// ----------------------------------------------------------
// PID01 spare
// ----------------------------------------------------------
// starting value -----------------------
//A     "U130ActD".Act.OutI // !!! insert correct Act !!!
      A     #GenRel;
      CLR   ;
      =     DB5306.DBX  203.2;
      =     DB5306.DBX  203.5;

// enable alarm -------------------------
      A     DB5306.DBX  203.5;
      A     DB5306.DBX  201.4;
      AN    DB5306.DBX  203.1;
      AN    DB5306.DBX  203.3;
      AN    DB5306.DBX  203.4;
      =     DB5306.DBX  203.0;

// setpoint to controller ---------------
      L     DB4301.DBD 1118; // !!! insert correct SFM !!!
      T     DB5306.DBD  234;

// static value to controller ----------
      L     DB4301.DBD 1118; // !!! insert correct SFM !!!
      T     DB5306.DBD  238;

// process value to controller ----------
      L     DB5303.DBD   26; // !!! insert correct AnI !!!
      T     DB5306.DBD  254;

// low/high value to controller ---------
      L     DB5303.DBD   30; // !!! insert correct AnI !!!
      T     DB5306.DBD  218;

      L     DB5303.DBD   34; // !!! insert correct AnI !!!
      T     DB5306.DBD  222;

NETWORK
TITLE =Sequence organisation

      CLR   ;
      =     M    122.2;

// SFM supply ----------------------------------------------------------------

// analog value to SFM spare -----------------------
      L     DB5303.DBD  146;
      T     DB4301.DBD 1122; // !!! insert correct SFM !!!

// analog value to SFM spare -----------------------
      L     DB5303.DBD  266;
      T     DB4301.DBD 1122; // !!! insert correct SFM !!!

// analog value to SFM spare -----------------------
      L     DB5303.DBD  386;
      T     DB4301.DBD 1122; // !!! insert correct SFM !!!

// sequencer ----------------------------------------------------------------
      A     DB4303.DBX   43.1;
      S     DB4303.DBX   97.3;

      CALL FC    40 (
           UnitNo                   := #UnitNo);

NETWORK
TITLE =Auto / Manual

      SET   ;
      AN    M    122.2;
      JC    MODE;
      AN    M    120.1;


// assign PID mode
      S     DB5306.DBX  201.4;
      S     DB5306.DBX  201.5;


MODE: SET   ;

END_FUNCTION_BLOCK

FUNCTION_BLOCK FB 4310
TITLE =U131: Planung Transfer J6F
FAMILY : BOTEC_F1
NAME : U131A
VERSION : 2.1


VAR_TEMP
  EStopOK : BOOL ;	//auxiliary flag
  CIP : BOOL ;	//CIP Program Selected
  xTmp : BOOL ;	//Temporary Bool(free for general use)
  DummyBool : BOOL ;	//Temporary Bool(free for general use)
  UnitNo : INT ;	//unit number
  UnitFB : INT ;	//unit expansion FB number
  rTmp : REAL ;	//Temporary REAL (free for general use)
  iTmp : INT ;	//Temporary INT (free for general use)
  DummyInt : INT ;	//Temporary INT (free for general use)
  dTmp : DINT ;	//Temporary DINT (free for general use)
END_VAR
BEGIN
NETWORK
TITLE =general

      CLR   ;
      =     #xTmp;
      =     #EStopOK;

      L     DB4310.DBW    0;
      T     #UnitNo;
      L     DB4310.DBW    2;
      T     #UnitFB;

NETWORK
TITLE =analog inputs

      NOP   0;
// C_AnI01 AnI 001 spare
      CALL FC    24 (
           UnitNo                   := #UnitNo,
           AnIRec                   := DB5313.C_AnI01,
           ValPer                   := #DummyInt);

// C_AnI002 AnI 002 spare
      CALL FC    24 (
           UnitNo                   := #UnitNo,
           AnIRec                   := DB5313.C_AnI002,
           ValPer                   := #DummyInt);

// AnI03 AnI 003 spare
      CALL FC    24 (
           UnitNo                   := #UnitNo,
           AnIRec                   := DB5313.AnI03,
           ValPer                   := #DummyInt);

NETWORK
TITLE =Universal value

      NOP   0;
// unv001 UnV 001 Process Status
      CALL FC    27 (
           UnitNo                   := #UnitNo,
           UnVRec                   := DB5315.unv001,
           ValExt                   := DB5315.DBD  234);

// unv002 UnV 002 Universal Value 02
      CALL FC    27 (
           UnitNo                   := #UnitNo,
           UnVRec                   := DB5315.unv002,
           ValExt                   := DB5315.DBD  362);

// unv003 UnV 003 Druck Sollwert
      CALL FC    27 (
           UnitNo                   := #UnitNo,
           UnVRec                   := DB5315.unv003,
           ValExt                   := DB5315.DBD  490);

// unv004 UnV 004 Universal Value 04
      CALL FC    27 (
           UnitNo                   := #UnitNo,
           UnVRec                   := DB5315.unv004,
           ValExt                   := DB5315.DBD  618);

NETWORK
TITLE =special inputs

      NOP   0;
// SpI01 SpI 001 spare
      CALL FC    14 (
           UnitNo                   := #UnitNo,
           SpIRec                   := DB5311.SpI01,
           SpIBit                   := #DummyBool);

// SpI02 SpI 002 spare
      CALL FC    14 (
           UnitNo                   := #UnitNo,
           SpIRec                   := DB5311.SpI02,
           SpIBit                   := #DummyBool);

// SpI03 SpI 003 spare
      CALL FC    14 (
           UnitNo                   := #UnitNo,
           SpIRec                   := DB5311.SpI03,
           SpIBit                   := #DummyBool);

// SpI04 SpI 004 spare
      CALL FC    14 (
           UnitNo                   := #UnitNo,
           SpIRec                   := DB5311.SpI04,
           SpIBit                   := #DummyBool);

NETWORK
TITLE =messages

      NOP   0;
// msg001 Msg 001 Message 01
      CALL FC    16 (
           UnitNo                   := #UnitNo,
           MsgRec                   := DB5317.msg001,
           MsgBit                   := DB5317.DBX   82.7);

// msg002 Msg 002 Message 02
      CALL FC    16 (
           UnitNo                   := #UnitNo,
           MsgRec                   := DB5317.msg002,
           MsgBit                   := DB5317.DBX  142.7);

// msg003 Msg 003 Message 03
      CALL FC    16 (
           UnitNo                   := #UnitNo,
           MsgRec                   := DB5317.msg003,
           MsgBit                   := DB5317.DBX  202.7);

NETWORK
TITLE =controllers

      NOP   0;
// PID01 PID 001 spare
      CALL FC    55 (
           UnitNo                   := #UnitNo,
           PIDRec                   := DB5316.PID01,
           SpExt                    := DB5316.DBD  234,
           PVal                     := DB5316.DBD  254,
           OPer                     := #DummyInt);

NETWORK
TITLE =unit supply

      UC    FB [#UnitFB];
END_FUNCTION_BLOCK

FUNCTION_BLOCK FB 4311
TITLE =U131: Planung Transfer J6F
FAMILY : BOTEC_F1
NAME : U131E
VERSION : 1.2


VAR_TEMP
  CIP : BOOL ;	//CIP active
  UNIM : BOOL ;	//Unit Not In Maintenance
  GenRel : BOOL ;	//general OK (emergency and maintenance OK)
  EStopOK : BOOL ;	//emergency OK
  UnitNo : INT ;	//unit number
  xTmp : BOOL ;	//Temporary Bool
  iTmp : INT ;	//Temporary INT
  rTmp : REAL ;	//Temporary REAL
  dTmp : DINT ;	//Temporary DINT (free for general use)
  RetValInt : INT ;	//return value
END_VAR
BEGIN
NETWORK
TITLE =General

      SET   ;
// Simulation ---------------------------------------------------------------
      A     DB4311.DBX 1357.7;
      CC    FB  4319; // "U131Sim"
      A     DB4311.DBX   17.3;
      =     DB4311.DBX 1357.7; //Help bit for simulation

// get unit number ----------------------------------------------------------
      L     DB4310.DBW    0;
      T     #UnitNo;

// CIP ----------------------------------------------------------------------
      L     DB4311.DBD   54;
      L     0;
      <D    ;
      =     #CIP;

// emergency OK -------------------------------------------------------------
      A     DB4315.DBX   27.0; //Emergency Stop OK
      =     #EStopOK;

// Write Unit in Maintenance ------------------------------------------------

      AN    DB4311.DBX   69.7;
      =     #UNIM;

// emergency and maintenance OK ---------------------------------------------
      A     #EStopOK;
      A     #UNIM;
      =     #GenRel;

// communication ------------------------------------------------------------
      UC    FB  4315; // U131Com

NETWORK
TITLE =Analog Inputs

      NOP   0;

// ----------------------------------------------------------
// C_AnI01 spare
// ----------------------------------------------------------
      L     DB4311.DBD 1118; // !!! insert correct SFM !!!
      T     DB5313.DBD  238;

      SET   ;
      =     DB5313.DBX  141.5;

// ----------------------------------------------------------
// C_AnI002 spare
// ----------------------------------------------------------
      L     DB4311.DBD 1118; // !!! insert correct SFM !!!
      T     DB5313.DBD  358;

      SET   ;
      =     DB5313.DBX  261.5;

// ----------------------------------------------------------
// AnI03 spare
// ----------------------------------------------------------
      L     DB4311.DBD 1118; // !!! insert correct SFM !!!
      T     DB5313.DBD  478;

      SET   ;
      =     DB5313.DBX  381.5;

NETWORK
TITLE =Universal Value

      NOP   0;

// ----------------------------------------------------------
// unv001 Process Status
// ----------------------------------------------------------
// process value to UnV
//      L     0.000000e+000
//      T     "U131UnVD".unv001.ValExt

// ----------------------------------------------------------
// unv002 Universal Value 02
// ----------------------------------------------------------
// process value to UnV
//      L     0.000000e+000
//      T     "U131UnVD".unv002.ValExt

// ----------------------------------------------------------
// unv003 Druck Sollwert
// ----------------------------------------------------------
// process value to UnV
//      L     0.000000e+000
//      T     "U131UnVD".unv003.ValExt

// ----------------------------------------------------------
// unv004 Universal Value 04
// ----------------------------------------------------------
// process value to UnV
//      L     0.000000e+000
//      T     "U131UnVD".unv004.ValExt

NETWORK
TITLE =Special Input

      NOP   0;

// ----------------------------------------------------------
// SpI01 spare
// ----------------------------------------------------------
      SET   ;
      =     DB5311.DBX   81.4;
      =     DB5311.DBX   81.5;

// ----------------------------------------------------------
// SpI02 spare
// ----------------------------------------------------------
      SET   ;
      =     DB5311.DBX  141.4;
      =     DB5311.DBX  141.5;

// ----------------------------------------------------------
// SpI03 spare
// ----------------------------------------------------------
      SET   ;
      =     DB5311.DBX  201.4;
      =     DB5311.DBX  201.5;

// ----------------------------------------------------------
// SpI04 spare
// ----------------------------------------------------------
      SET   ;
      =     DB5311.DBX  261.4;
      =     DB5311.DBX  261.5;

NETWORK
TITLE =Messages

      NOP   0;

// ----------------------------------------------------------
// msg001 Message 01
// ----------------------------------------------------------
      SET   ;
      R     DB5317.DBX   80.7;
      =     DB5317.DBX   81.4;

      CLR   ;
      =     DB5317.DBX   82.7;

// ----------------------------------------------------------
// msg002 Message 02
// ----------------------------------------------------------
      SET   ;
      R     DB5317.DBX  140.7;
      =     DB5317.DBX  141.4;

      CLR   ;
      =     DB5317.DBX  142.7;

// ----------------------------------------------------------
// msg003 Message 03
// ----------------------------------------------------------
      SET   ;
      R     DB5317.DBX  200.7;
      =     DB5317.DBX  201.4;

      CLR   ;
      =     DB5317.DBX  202.7;

NETWORK
TITLE =PID controller

      NOP   0;

// ----------------------------------------------------------
// PID01 spare
// ----------------------------------------------------------
// starting value -----------------------
//A     "U131ActD".Act.OutI // !!! insert correct Act !!!
      A     #GenRel;
      CLR   ;
      =     DB5316.DBX  203.2;
      =     DB5316.DBX  203.5;

// enable alarm -------------------------
      A     DB5316.DBX  203.5;
      A     DB5316.DBX  201.4;
      AN    DB5316.DBX  203.1;
      AN    DB5316.DBX  203.3;
      AN    DB5316.DBX  203.4;
      =     DB5316.DBX  203.0;

// setpoint to controller ---------------
      L     DB4311.DBD 1118; // !!! insert correct SFM !!!
      T     DB5316.DBD  234;

// static value to controller ----------
      L     DB4311.DBD 1118; // !!! insert correct SFM !!!
      T     DB5316.DBD  238;

// process value to controller ----------
      L     DB5313.DBD   26; // !!! insert correct AnI !!!
      T     DB5316.DBD  254;

// low/high value to controller ---------
      L     DB5313.DBD   30; // !!! insert correct AnI !!!
      T     DB5316.DBD  218;

      L     DB5313.DBD   34; // !!! insert correct AnI !!!
      T     DB5316.DBD  222;

NETWORK
TITLE =Sequence organisation

      CLR   ;
      =     M    122.2;

// SFM supply ----------------------------------------------------------------

// analog value to SFM spare -----------------------
      L     DB5313.DBD  146;
      T     DB4311.DBD 1122; // !!! insert correct SFM !!!

// analog value to SFM spare -----------------------
      L     DB5313.DBD  266;
      T     DB4311.DBD 1122; // !!! insert correct SFM !!!

// analog value to SFM spare -----------------------
      L     DB5313.DBD  386;
      T     DB4311.DBD 1122; // !!! insert correct SFM !!!

// sequencer ----------------------------------------------------------------
      A     DB4313.DBX   43.1;
      S     DB4313.DBX   97.3;

      CALL FC    40 (
           UnitNo                   := #UnitNo);

NETWORK
TITLE =Auto / Manual

      SET   ;
      AN    M    122.2;
      JC    MODE;
      AN    M    120.1;


// assign PID mode
      S     DB5316.DBX  201.4;
      S     DB5316.DBX  201.5;


MODE: SET   ;

END_FUNCTION_BLOCK

FUNCTION_BLOCK FB 4320
TITLE =U132: Planung Transfer L6F
FAMILY : BOTEC_F1
NAME : U132A
VERSION : 2.1


VAR_TEMP
  EStopOK : BOOL ;	//auxiliary flag
  CIP : BOOL ;	//CIP Program Selected
  xTmp : BOOL ;	//Temporary Bool(free for general use)
  DummyBool : BOOL ;	//Temporary Bool(free for general use)
  UnitNo : INT ;	//unit number
  UnitFB : INT ;	//unit expansion FB number
  rTmp : REAL ;	//Temporary REAL (free for general use)
  iTmp : INT ;	//Temporary INT (free for general use)
  DummyInt : INT ;	//Temporary INT (free for general use)
  dTmp : DINT ;	//Temporary DINT (free for general use)
END_VAR
BEGIN
NETWORK
TITLE =general

      CLR   ;
      =     #xTmp;
      =     #EStopOK;

      L     DB4320.DBW    0;
      T     #UnitNo;
      L     DB4320.DBW    2;
      T     #UnitFB;

NETWORK
TITLE =analog inputs

      NOP   0;
// C_AnI01 AnI 001 spare
      CALL FC    24 (
           UnitNo                   := #UnitNo,
           AnIRec                   := DB5323.C_AnI01,
           ValPer                   := #DummyInt);

// C_AnI002 AnI 002 spare
      CALL FC    24 (
           UnitNo                   := #UnitNo,
           AnIRec                   := DB5323.C_AnI002,
           ValPer                   := #DummyInt);

// AnI03 AnI 003 spare
      CALL FC    24 (
           UnitNo                   := #UnitNo,
           AnIRec                   := DB5323.AnI03,
           ValPer                   := #DummyInt);

NETWORK
TITLE =Universal value

      NOP   0;
// unv001 UnV 001 Process Status
      CALL FC    27 (
           UnitNo                   := #UnitNo,
           UnVRec                   := DB5325.unv001,
           ValExt                   := DB5325.DBD  234);

// unv002 UnV 002 Universal Value 02
      CALL FC    27 (
           UnitNo                   := #UnitNo,
           UnVRec                   := DB5325.unv002,
           ValExt                   := DB5325.DBD  362);

// unv003 UnV 003 Druck Sollwert
      CALL FC    27 (
           UnitNo                   := #UnitNo,
           UnVRec                   := DB5325.unv003,
           ValExt                   := DB5325.DBD  490);

// unv004 UnV 004 Universal Value 04
      CALL FC    27 (
           UnitNo                   := #UnitNo,
           UnVRec                   := DB5325.unv004,
           ValExt                   := DB5325.DBD  618);

NETWORK
TITLE =special inputs

      NOP   0;
// SpI01 SpI 001 spare
      CALL FC    14 (
           UnitNo                   := #UnitNo,
           SpIRec                   := DB5321.SpI01,
           SpIBit                   := #DummyBool);

// SpI02 SpI 002 spare
      CALL FC    14 (
           UnitNo                   := #UnitNo,
           SpIRec                   := DB5321.SpI02,
           SpIBit                   := #DummyBool);

// SpI03 SpI 003 spare
      CALL FC    14 (
           UnitNo                   := #UnitNo,
           SpIRec                   := DB5321.SpI03,
           SpIBit                   := #DummyBool);

// SpI04 SpI 004 spare
      CALL FC    14 (
           UnitNo                   := #UnitNo,
           SpIRec                   := DB5321.SpI04,
           SpIBit                   := #DummyBool);

NETWORK
TITLE =messages

      NOP   0;
// msg001 Msg 001 Message 01
      CALL FC    16 (
           UnitNo                   := #UnitNo,
           MsgRec                   := DB5327.msg001,
           MsgBit                   := DB5327.DBX   82.7);

// msg002 Msg 002 Message 02
      CALL FC    16 (
           UnitNo                   := #UnitNo,
           MsgRec                   := DB5327.msg002,
           MsgBit                   := DB5327.DBX  142.7);

// msg003 Msg 003 Message 03
      CALL FC    16 (
           UnitNo                   := #UnitNo,
           MsgRec                   := DB5327.msg003,
           MsgBit                   := DB5327.DBX  202.7);

NETWORK
TITLE =controllers

      NOP   0;
// PID01 PID 001 spare
      CALL FC    55 (
           UnitNo                   := #UnitNo,
           PIDRec                   := DB5326.PID01,
           SpExt                    := DB5326.DBD  234,
           PVal                     := DB5326.DBD  254,
           OPer                     := #DummyInt);

NETWORK
TITLE =unit supply

      UC    FB [#UnitFB];
END_FUNCTION_BLOCK

FUNCTION_BLOCK FB 4321
TITLE =U132: Planung Transfer L6F
FAMILY : BOTEC_F1
NAME : U132E
VERSION : 1.2


VAR_TEMP
  CIP : BOOL ;	//CIP active
  UNIM : BOOL ;	//Unit Not In Maintenance
  GenRel : BOOL ;	//general OK (emergency and maintenance OK)
  EStopOK : BOOL ;	//emergency OK
  UnitNo : INT ;	//unit number
  xTmp : BOOL ;	//Temporary Bool
  iTmp : INT ;	//Temporary INT
  rTmp : REAL ;	//Temporary REAL
  dTmp : DINT ;	//Temporary DINT (free for general use)
  RetValInt : INT ;	//return value
END_VAR
BEGIN
NETWORK
TITLE =General

      SET   ;
// Simulation ---------------------------------------------------------------
      A     DB4321.DBX 1357.7;
      CC    FB  4329; // "U132Sim"
      A     DB4321.DBX   17.3;
      =     DB4321.DBX 1357.7; //Help bit for simulation

// get unit number ----------------------------------------------------------
      L     DB4320.DBW    0;
      T     #UnitNo;

// CIP ----------------------------------------------------------------------
      L     DB4321.DBD   54;
      L     0;
      <D    ;
      =     #CIP;

// emergency OK -------------------------------------------------------------
      A     DB4325.DBX   27.0; //Emergency Stop OK
      =     #EStopOK;

// Write Unit in Maintenance ------------------------------------------------

      AN    DB4321.DBX   69.7;
      =     #UNIM;

// emergency and maintenance OK ---------------------------------------------
      A     #EStopOK;
      A     #UNIM;
      =     #GenRel;

// communication ------------------------------------------------------------
      UC    FB  4325; // U132Com

NETWORK
TITLE =Analog Inputs

      NOP   0;

// ----------------------------------------------------------
// C_AnI01 spare
// ----------------------------------------------------------
      L     DB4321.DBD 1118; // !!! insert correct SFM !!!
      T     DB5323.DBD  238;

      SET   ;
      =     DB5323.DBX  141.5;

// ----------------------------------------------------------
// C_AnI002 spare
// ----------------------------------------------------------
      L     DB4321.DBD 1118; // !!! insert correct SFM !!!
      T     DB5323.DBD  358;

      SET   ;
      =     DB5323.DBX  261.5;

// ----------------------------------------------------------
// AnI03 spare
// ----------------------------------------------------------
      L     DB4321.DBD 1118; // !!! insert correct SFM !!!
      T     DB5323.DBD  478;

      SET   ;
      =     DB5323.DBX  381.5;

NETWORK
TITLE =Universal Value

      NOP   0;

// ----------------------------------------------------------
// unv001 Process Status
// ----------------------------------------------------------
// process value to UnV
//      L     0.000000e+000
//      T     "U132UnVD".unv001.ValExt

// ----------------------------------------------------------
// unv002 Universal Value 02
// ----------------------------------------------------------
// process value to UnV
//      L     0.000000e+000
//      T     "U132UnVD".unv002.ValExt

// ----------------------------------------------------------
// unv003 Druck Sollwert
// ----------------------------------------------------------
// process value to UnV
//      L     0.000000e+000
//      T     "U132UnVD".unv003.ValExt

// ----------------------------------------------------------
// unv004 Universal Value 04
// ----------------------------------------------------------
// process value to UnV
//      L     0.000000e+000
//      T     "U132UnVD".unv004.ValExt

NETWORK
TITLE =Special Input

      NOP   0;

// ----------------------------------------------------------
// SpI01 spare
// ----------------------------------------------------------
      SET   ;
      =     DB5321.DBX   81.4;
      =     DB5321.DBX   81.5;

// ----------------------------------------------------------
// SpI02 spare
// ----------------------------------------------------------
      SET   ;
      =     DB5321.DBX  141.4;
      =     DB5321.DBX  141.5;

// ----------------------------------------------------------
// SpI03 spare
// ----------------------------------------------------------
      SET   ;
      =     DB5321.DBX  201.4;
      =     DB5321.DBX  201.5;

// ----------------------------------------------------------
// SpI04 spare
// ----------------------------------------------------------
      SET   ;
      =     DB5321.DBX  261.4;
      =     DB5321.DBX  261.5;

NETWORK
TITLE =Messages

      NOP   0;

// ----------------------------------------------------------
// msg001 Message 01
// ----------------------------------------------------------
      SET   ;
      R     DB5327.DBX   80.7;
      =     DB5327.DBX   81.4;

      CLR   ;
      =     DB5327.DBX   82.7;

// ----------------------------------------------------------
// msg002 Message 02
// ----------------------------------------------------------
      SET   ;
      R     DB5327.DBX  140.7;
      =     DB5327.DBX  141.4;

      CLR   ;
      =     DB5327.DBX  142.7;

// ----------------------------------------------------------
// msg003 Message 03
// ----------------------------------------------------------
      SET   ;
      R     DB5327.DBX  200.7;
      =     DB5327.DBX  201.4;

      CLR   ;
      =     DB5327.DBX  202.7;

NETWORK
TITLE =PID controller

      NOP   0;

// ----------------------------------------------------------
// PID01 spare
// ----------------------------------------------------------
// starting value -----------------------
//A     "U132ActD".Act.OutI // !!! insert correct Act !!!
      A     #GenRel;
      CLR   ;
      =     DB5326.DBX  203.2;
      =     DB5326.DBX  203.5;

// enable alarm -------------------------
      A     DB5326.DBX  203.5;
      A     DB5326.DBX  201.4;
      AN    DB5326.DBX  203.1;
      AN    DB5326.DBX  203.3;
      AN    DB5326.DBX  203.4;
      =     DB5326.DBX  203.0;

// setpoint to controller ---------------
      L     DB4321.DBD 1118; // !!! insert correct SFM !!!
      T     DB5326.DBD  234;

// static value to controller ----------
      L     DB4321.DBD 1118; // !!! insert correct SFM !!!
      T     DB5326.DBD  238;

// process value to controller ----------
      L     DB5323.DBD   26; // !!! insert correct AnI !!!
      T     DB5326.DBD  254;

// low/high value to controller ---------
      L     DB5323.DBD   30; // !!! insert correct AnI !!!
      T     DB5326.DBD  218;

      L     DB5323.DBD   34; // !!! insert correct AnI !!!
      T     DB5326.DBD  222;

NETWORK
TITLE =Sequence organisation

      CLR   ;
      =     M    122.2;

// SFM supply ----------------------------------------------------------------

// analog value to SFM spare -----------------------
      L     DB5323.DBD  146;
      T     DB4321.DBD 1122; // !!! insert correct SFM !!!

// analog value to SFM spare -----------------------
      L     DB5323.DBD  266;
      T     DB4321.DBD 1122; // !!! insert correct SFM !!!

// analog value to SFM spare -----------------------
      L     DB5323.DBD  386;
      T     DB4321.DBD 1122; // !!! insert correct SFM !!!

// sequencer ----------------------------------------------------------------
      A     DB4323.DBX   43.1;
      S     DB4323.DBX   97.3;

      CALL FC    40 (
           UnitNo                   := #UnitNo);

NETWORK
TITLE =Auto / Manual

      SET   ;
      AN    M    122.2;
      JC    MODE;
      AN    M    120.1;


// assign PID mode
      S     DB5326.DBX  201.4;
      S     DB5326.DBX  201.5;


MODE: SET   ;

END_FUNCTION_BLOCK

FUNCTION_BLOCK FB 4330
TITLE =U133: Planung Transfer B6
FAMILY : BOTEC_F1
NAME : U133A
VERSION : 2.1


VAR_TEMP
  EStopOK : BOOL ;	//auxiliary flag
  CIP : BOOL ;	//CIP Program Selected
  xTmp : BOOL ;	//Temporary Bool(free for general use)
  DummyBool : BOOL ;	//Temporary Bool(free for general use)
  UnitNo : INT ;	//unit number
  UnitFB : INT ;	//unit expansion FB number
  rTmp : REAL ;	//Temporary REAL (free for general use)
  iTmp : INT ;	//Temporary INT (free for general use)
  DummyInt : INT ;	//Temporary INT (free for general use)
  dTmp : DINT ;	//Temporary DINT (free for general use)
END_VAR
BEGIN
NETWORK
TITLE =general

      CLR   ;
      =     #xTmp;
      =     #EStopOK;

      L     DB4330.DBW    0;
      T     #UnitNo;
      L     DB4330.DBW    2;
      T     #UnitFB;

NETWORK
TITLE =analog inputs

      NOP   0;
// C_AnI01 AnI 001 spare
      CALL FC    24 (
           UnitNo                   := #UnitNo,
           AnIRec                   := DB5333.C_AnI01,
           ValPer                   := #DummyInt);

// C_AnI002 AnI 002 spare
      CALL FC    24 (
           UnitNo                   := #UnitNo,
           AnIRec                   := DB5333.C_AnI002,
           ValPer                   := #DummyInt);

// AnI03 AnI 003 spare
      CALL FC    24 (
           UnitNo                   := #UnitNo,
           AnIRec                   := DB5333.AnI03,
           ValPer                   := #DummyInt);

NETWORK
TITLE =Universal value

      NOP   0;
// unv001 UnV 001 Process Status
      CALL FC    27 (
           UnitNo                   := #UnitNo,
           UnVRec                   := DB5335.unv001,
           ValExt                   := DB5335.DBD  234);

// unv002 UnV 002 Universal Value 02
      CALL FC    27 (
           UnitNo                   := #UnitNo,
           UnVRec                   := DB5335.unv002,
           ValExt                   := DB5335.DBD  362);

// unv003 UnV 003 Druck Sollwert
      CALL FC    27 (
           UnitNo                   := #UnitNo,
           UnVRec                   := DB5335.unv003,
           ValExt                   := DB5335.DBD  490);

// unv004 UnV 004 Universal Value 04
      CALL FC    27 (
           UnitNo                   := #UnitNo,
           UnVRec                   := DB5335.unv004,
           ValExt                   := DB5335.DBD  618);

NETWORK
TITLE =special inputs

      NOP   0;
// SpI01 SpI 001 spare
      CALL FC    14 (
           UnitNo                   := #UnitNo,
           SpIRec                   := DB5331.SpI01,
           SpIBit                   := #DummyBool);

// SpI02 SpI 002 spare
      CALL FC    14 (
           UnitNo                   := #UnitNo,
           SpIRec                   := DB5331.SpI02,
           SpIBit                   := #DummyBool);

// SpI03 SpI 003 spare
      CALL FC    14 (
           UnitNo                   := #UnitNo,
           SpIRec                   := DB5331.SpI03,
           SpIBit                   := #DummyBool);

// SpI04 SpI 004 spare
      CALL FC    14 (
           UnitNo                   := #UnitNo,
           SpIRec                   := DB5331.SpI04,
           SpIBit                   := #DummyBool);

NETWORK
TITLE =messages

      NOP   0;
// msg001 Msg 001 Message 01
      CALL FC    16 (
           UnitNo                   := #UnitNo,
           MsgRec                   := DB5337.msg001,
           MsgBit                   := DB5337.DBX   82.7);

// msg002 Msg 002 Message 02
      CALL FC    16 (
           UnitNo                   := #UnitNo,
           MsgRec                   := DB5337.msg002,
           MsgBit                   := DB5337.DBX  142.7);

// msg003 Msg 003 Message 03
      CALL FC    16 (
           UnitNo                   := #UnitNo,
           MsgRec                   := DB5337.msg003,
           MsgBit                   := DB5337.DBX  202.7);

NETWORK
TITLE =controllers

      NOP   0;
// PID01 PID 001 spare
      CALL FC    55 (
           UnitNo                   := #UnitNo,
           PIDRec                   := DB5336.PID01,
           SpExt                    := DB5336.DBD  234,
           PVal                     := DB5336.DBD  254,
           OPer                     := #DummyInt);

NETWORK
TITLE =unit supply

      UC    FB [#UnitFB];
END_FUNCTION_BLOCK

FUNCTION_BLOCK FB 4331
TITLE =U133: Planung Transfer B6
FAMILY : BOTEC_F1
NAME : U133E
VERSION : 1.2


VAR_TEMP
  CIP : BOOL ;	//CIP active
  UNIM : BOOL ;	//Unit Not In Maintenance
  GenRel : BOOL ;	//general OK (emergency and maintenance OK)
  EStopOK : BOOL ;	//emergency OK
  UnitNo : INT ;	//unit number
  xTmp : BOOL ;	//Temporary Bool
  iTmp : INT ;	//Temporary INT
  rTmp : REAL ;	//Temporary REAL
  dTmp : DINT ;	//Temporary DINT (free for general use)
  RetValInt : INT ;	//return value
END_VAR
BEGIN
NETWORK
TITLE =General

      SET   ;
// Simulation ---------------------------------------------------------------
      A     DB4331.DBX 1357.7;
      CC    FB  4339; // "U133Sim"
      A     DB4331.DBX   17.3;
      =     DB4331.DBX 1357.7; //Help bit for simulation

// get unit number ----------------------------------------------------------
      L     DB4330.DBW    0;
      T     #UnitNo;

// CIP ----------------------------------------------------------------------
      L     DB4331.DBD   54;
      L     0;
      <D    ;
      =     #CIP;

// emergency OK -------------------------------------------------------------
      A     DB4335.DBX   27.0; //Emergency Stop OK
      =     #EStopOK;

// Write Unit in Maintenance ------------------------------------------------

      AN    DB4331.DBX   69.7;
      =     #UNIM;

// emergency and maintenance OK ---------------------------------------------
      A     #EStopOK;
      A     #UNIM;
      =     #GenRel;

// communication ------------------------------------------------------------
      UC    FB  4335; // U133Com

NETWORK
TITLE =Analog Inputs

      NOP   0;

// ----------------------------------------------------------
// C_AnI01 spare
// ----------------------------------------------------------
      L     DB4331.DBD 1118; // !!! insert correct SFM !!!
      T     DB5333.DBD  238;

      SET   ;
      =     DB5333.DBX  141.5;

// ----------------------------------------------------------
// C_AnI002 spare
// ----------------------------------------------------------
      L     DB4331.DBD 1118; // !!! insert correct SFM !!!
      T     DB5333.DBD  358;

      SET   ;
      =     DB5333.DBX  261.5;

// ----------------------------------------------------------
// AnI03 spare
// ----------------------------------------------------------
      L     DB4331.DBD 1118; // !!! insert correct SFM !!!
      T     DB5333.DBD  478;

      SET   ;
      =     DB5333.DBX  381.5;

NETWORK
TITLE =Universal Value

      NOP   0;

// ----------------------------------------------------------
// unv001 Process Status
// ----------------------------------------------------------
// process value to UnV
//      L     0.000000e+000
//      T     "U133UnVD".unv001.ValExt

// ----------------------------------------------------------
// unv002 Universal Value 02
// ----------------------------------------------------------
// process value to UnV
//      L     0.000000e+000
//      T     "U133UnVD".unv002.ValExt

// ----------------------------------------------------------
// unv003 Druck Sollwert
// ----------------------------------------------------------
// process value to UnV
//      L     0.000000e+000
//      T     "U133UnVD".unv003.ValExt

// ----------------------------------------------------------
// unv004 Universal Value 04
// ----------------------------------------------------------
// process value to UnV
//      L     0.000000e+000
//      T     "U133UnVD".unv004.ValExt

NETWORK
TITLE =Special Input

      NOP   0;

// ----------------------------------------------------------
// SpI01 spare
// ----------------------------------------------------------
      SET   ;
      =     DB5331.DBX   81.4;
      =     DB5331.DBX   81.5;

// ----------------------------------------------------------
// SpI02 spare
// ----------------------------------------------------------
      SET   ;
      =     DB5331.DBX  141.4;
      =     DB5331.DBX  141.5;

// ----------------------------------------------------------
// SpI03 spare
// ----------------------------------------------------------
      SET   ;
      =     DB5331.DBX  201.4;
      =     DB5331.DBX  201.5;

// ----------------------------------------------------------
// SpI04 spare
// ----------------------------------------------------------
      SET   ;
      =     DB5331.DBX  261.4;
      =     DB5331.DBX  261.5;

NETWORK
TITLE =Messages

      NOP   0;

// ----------------------------------------------------------
// msg001 Message 01
// ----------------------------------------------------------
      SET   ;
      R     DB5337.DBX   80.7;
      =     DB5337.DBX   81.4;

      CLR   ;
      =     DB5337.DBX   82.7;

// ----------------------------------------------------------
// msg002 Message 02
// ----------------------------------------------------------
      SET   ;
      R     DB5337.DBX  140.7;
      =     DB5337.DBX  141.4;

      CLR   ;
      =     DB5337.DBX  142.7;

// ----------------------------------------------------------
// msg003 Message 03
// ----------------------------------------------------------
      SET   ;
      R     DB5337.DBX  200.7;
      =     DB5337.DBX  201.4;

      CLR   ;
      =     DB5337.DBX  202.7;

NETWORK
TITLE =PID controller

      NOP   0;

// ----------------------------------------------------------
// PID01 spare
// ----------------------------------------------------------
// starting value -----------------------
//A     "U133ActD".Act.OutI // !!! insert correct Act !!!
      A     #GenRel;
      CLR   ;
      =     DB5336.DBX  203.2;
      =     DB5336.DBX  203.5;

// enable alarm -------------------------
      A     DB5336.DBX  203.5;
      A     DB5336.DBX  201.4;
      AN    DB5336.DBX  203.1;
      AN    DB5336.DBX  203.3;
      AN    DB5336.DBX  203.4;
      =     DB5336.DBX  203.0;

// setpoint to controller ---------------
      L     DB4331.DBD 1118; // !!! insert correct SFM !!!
      T     DB5336.DBD  234;

// static value to controller ----------
      L     DB4331.DBD 1118; // !!! insert correct SFM !!!
      T     DB5336.DBD  238;

// process value to controller ----------
      L     DB5333.DBD   26; // !!! insert correct AnI !!!
      T     DB5336.DBD  254;

// low/high value to controller ---------
      L     DB5333.DBD   30; // !!! insert correct AnI !!!
      T     DB5336.DBD  218;

      L     DB5333.DBD   34; // !!! insert correct AnI !!!
      T     DB5336.DBD  222;

NETWORK
TITLE =Sequence organisation

      CLR   ;
      =     M    122.2;

// SFM supply ----------------------------------------------------------------

// analog value to SFM spare -----------------------
      L     DB5333.DBD  146;
      T     DB4331.DBD 1122; // !!! insert correct SFM !!!

// analog value to SFM spare -----------------------
      L     DB5333.DBD  266;
      T     DB4331.DBD 1122; // !!! insert correct SFM !!!

// analog value to SFM spare -----------------------
      L     DB5333.DBD  386;
      T     DB4331.DBD 1122; // !!! insert correct SFM !!!

// sequencer ----------------------------------------------------------------
      A     DB4333.DBX   43.1;
      S     DB4333.DBX   97.3;

      CALL FC    40 (
           UnitNo                   := #UnitNo);

NETWORK
TITLE =Auto / Manual

      SET   ;
      AN    M    122.2;
      JC    MODE;
      AN    M    120.1;


// assign PID mode
      S     DB5336.DBX  201.4;
      S     DB5336.DBX  201.5;


MODE: SET   ;

END_FUNCTION_BLOCK

FUNCTION_BLOCK FB 4340
TITLE =U134: Planung Transfer D6
FAMILY : BOTEC_F1
NAME : U134A
VERSION : 2.1


VAR_TEMP
  EStopOK : BOOL ;	//auxiliary flag
  CIP : BOOL ;	//CIP Program Selected
  xTmp : BOOL ;	//Temporary Bool(free for general use)
  DummyBool : BOOL ;	//Temporary Bool(free for general use)
  UnitNo : INT ;	//unit number
  UnitFB : INT ;	//unit expansion FB number
  rTmp : REAL ;	//Temporary REAL (free for general use)
  iTmp : INT ;	//Temporary INT (free for general use)
  DummyInt : INT ;	//Temporary INT (free for general use)
  dTmp : DINT ;	//Temporary DINT (free for general use)
END_VAR
BEGIN
NETWORK
TITLE =general

      CLR   ;
      =     #xTmp;
      =     #EStopOK;

      L     DB4340.DBW    0;
      T     #UnitNo;
      L     DB4340.DBW    2;
      T     #UnitFB;

NETWORK
TITLE =analog inputs

      NOP   0;
// C_AnI01 AnI 001 spare
      CALL FC    24 (
           UnitNo                   := #UnitNo,
           AnIRec                   := DB5343.C_AnI01,
           ValPer                   := #DummyInt);

// C_AnI002 AnI 002 spare
      CALL FC    24 (
           UnitNo                   := #UnitNo,
           AnIRec                   := DB5343.C_AnI002,
           ValPer                   := #DummyInt);

// AnI03 AnI 003 spare
      CALL FC    24 (
           UnitNo                   := #UnitNo,
           AnIRec                   := DB5343.AnI03,
           ValPer                   := #DummyInt);

NETWORK
TITLE =Universal value

      NOP   0;
// unv001 UnV 001 Process Status
      CALL FC    27 (
           UnitNo                   := #UnitNo,
           UnVRec                   := DB5345.unv001,
           ValExt                   := DB5345.DBD  234);

// unv002 UnV 002 Universal Value 02
      CALL FC    27 (
           UnitNo                   := #UnitNo,
           UnVRec                   := DB5345.unv002,
           ValExt                   := DB5345.DBD  362);

// unv003 UnV 003 Druck Sollwert
      CALL FC    27 (
           UnitNo                   := #UnitNo,
           UnVRec                   := DB5345.unv003,
           ValExt                   := DB5345.DBD  490);

// unv004 UnV 004 Universal Value 04
      CALL FC    27 (
           UnitNo                   := #UnitNo,
           UnVRec                   := DB5345.unv004,
           ValExt                   := DB5345.DBD  618);

NETWORK
TITLE =special inputs

      NOP   0;
// SpI01 SpI 001 spare
      CALL FC    14 (
           UnitNo                   := #UnitNo,
           SpIRec                   := DB5341.SpI01,
           SpIBit                   := #DummyBool);

// SpI02 SpI 002 spare
      CALL FC    14 (
           UnitNo                   := #UnitNo,
           SpIRec                   := DB5341.SpI02,
           SpIBit                   := #DummyBool);

// SpI03 SpI 003 spare
      CALL FC    14 (
           UnitNo                   := #UnitNo,
           SpIRec                   := DB5341.SpI03,
           SpIBit                   := #DummyBool);

// SpI04 SpI 004 spare
      CALL FC    14 (
           UnitNo                   := #UnitNo,
           SpIRec                   := DB5341.SpI04,
           SpIBit                   := #DummyBool);

NETWORK
TITLE =messages

      NOP   0;
// msg001 Msg 001 Message 01
      CALL FC    16 (
           UnitNo                   := #UnitNo,
           MsgRec                   := DB5347.msg001,
           MsgBit                   := DB5347.DBX   82.7);

// msg002 Msg 002 Message 02
      CALL FC    16 (
           UnitNo                   := #UnitNo,
           MsgRec                   := DB5347.msg002,
           MsgBit                   := DB5347.DBX  142.7);

// msg003 Msg 003 Message 03
      CALL FC    16 (
           UnitNo                   := #UnitNo,
           MsgRec                   := DB5347.msg003,
           MsgBit                   := DB5347.DBX  202.7);

NETWORK
TITLE =controllers

      NOP   0;
// PID01 PID 001 spare
      CALL FC    55 (
           UnitNo                   := #UnitNo,
           PIDRec                   := DB5346.PID01,
           SpExt                    := DB5346.DBD  234,
           PVal                     := DB5346.DBD  254,
           OPer                     := #DummyInt);

NETWORK
TITLE =unit supply

      UC    FB [#UnitFB];
END_FUNCTION_BLOCK

FUNCTION_BLOCK FB 4341
TITLE =U134: Planung Transfer D6
FAMILY : BOTEC_F1
NAME : U134E
VERSION : 1.2


VAR_TEMP
  CIP : BOOL ;	//CIP active
  UNIM : BOOL ;	//Unit Not In Maintenance
  GenRel : BOOL ;	//general OK (emergency and maintenance OK)
  EStopOK : BOOL ;	//emergency OK
  UnitNo : INT ;	//unit number
  xTmp : BOOL ;	//Temporary Bool
  iTmp : INT ;	//Temporary INT
  rTmp : REAL ;	//Temporary REAL
  dTmp : DINT ;	//Temporary DINT (free for general use)
  RetValInt : INT ;	//return value
END_VAR
BEGIN
NETWORK
TITLE =General

      SET   ;
// Simulation ---------------------------------------------------------------
      A     DB4341.DBX 1357.7;
      CC    FB  4349; // "U134Sim"
      A     DB4341.DBX   17.3;
      =     DB4341.DBX 1357.7; //Help bit for simulation

// get unit number ----------------------------------------------------------
      L     DB4340.DBW    0;
      T     #UnitNo;

// CIP ----------------------------------------------------------------------
      L     DB4341.DBD   54;
      L     0;
      <D    ;
      =     #CIP;

// emergency OK -------------------------------------------------------------
      A     DB4345.DBX   27.0; //Emergency Stop OK
      =     #EStopOK;

// Write Unit in Maintenance ------------------------------------------------

      AN    DB4341.DBX   69.7;
      =     #UNIM;

// emergency and maintenance OK ---------------------------------------------
      A     #EStopOK;
      A     #UNIM;
      =     #GenRel;

// communication ------------------------------------------------------------
      UC    FB  4345; // U134Com

NETWORK
TITLE =Analog Inputs

      NOP   0;

// ----------------------------------------------------------
// C_AnI01 spare
// ----------------------------------------------------------
      L     DB4341.DBD 1118; // !!! insert correct SFM !!!
      T     DB5343.DBD  238;

      SET   ;
      =     DB5343.DBX  141.5;

// ----------------------------------------------------------
// C_AnI002 spare
// ----------------------------------------------------------
      L     DB4341.DBD 1118; // !!! insert correct SFM !!!
      T     DB5343.DBD  358;

      SET   ;
      =     DB5343.DBX  261.5;

// ----------------------------------------------------------
// AnI03 spare
// ----------------------------------------------------------
      L     DB4341.DBD 1118; // !!! insert correct SFM !!!
      T     DB5343.DBD  478;

      SET   ;
      =     DB5343.DBX  381.5;

NETWORK
TITLE =Universal Value

      NOP   0;

// ----------------------------------------------------------
// unv001 Process Status
// ----------------------------------------------------------
// process value to UnV
//      L     0.000000e+000
//      T     "U134UnVD".unv001.ValExt

// ----------------------------------------------------------
// unv002 Universal Value 02
// ----------------------------------------------------------
// process value to UnV
//      L     0.000000e+000
//      T     "U134UnVD".unv002.ValExt

// ----------------------------------------------------------
// unv003 Druck Sollwert
// ----------------------------------------------------------
// process value to UnV
//      L     0.000000e+000
//      T     "U134UnVD".unv003.ValExt

// ----------------------------------------------------------
// unv004 Universal Value 04
// ----------------------------------------------------------
// process value to UnV
//      L     0.000000e+000
//      T     "U134UnVD".unv004.ValExt

NETWORK
TITLE =Special Input

      NOP   0;

// ----------------------------------------------------------
// SpI01 spare
// ----------------------------------------------------------
      SET   ;
      =     DB5341.DBX   81.4;
      =     DB5341.DBX   81.5;

// ----------------------------------------------------------
// SpI02 spare
// ----------------------------------------------------------
      SET   ;
      =     DB5341.DBX  141.4;
      =     DB5341.DBX  141.5;

// ----------------------------------------------------------
// SpI03 spare
// ----------------------------------------------------------
      SET   ;
      =     DB5341.DBX  201.4;
      =     DB5341.DBX  201.5;

// ----------------------------------------------------------
// SpI04 spare
// ----------------------------------------------------------
      SET   ;
      =     DB5341.DBX  261.4;
      =     DB5341.DBX  261.5;

NETWORK
TITLE =Messages

      NOP   0;

// ----------------------------------------------------------
// msg001 Message 01
// ----------------------------------------------------------
      SET   ;
      R     DB5347.DBX   80.7;
      =     DB5347.DBX   81.4;

      CLR   ;
      =     DB5347.DBX   82.7;

// ----------------------------------------------------------
// msg002 Message 02
// ----------------------------------------------------------
      SET   ;
      R     DB5347.DBX  140.7;
      =     DB5347.DBX  141.4;

      CLR   ;
      =     DB5347.DBX  142.7;

// ----------------------------------------------------------
// msg003 Message 03
// ----------------------------------------------------------
      SET   ;
      R     DB5347.DBX  200.7;
      =     DB5347.DBX  201.4;

      CLR   ;
      =     DB5347.DBX  202.7;

NETWORK
TITLE =PID controller

      NOP   0;

// ----------------------------------------------------------
// PID01 spare
// ----------------------------------------------------------
// starting value -----------------------
//A     "U134ActD".Act.OutI // !!! insert correct Act !!!
      A     #GenRel;
      CLR   ;
      =     DB5346.DBX  203.2;
      =     DB5346.DBX  203.5;

// enable alarm -------------------------
      A     DB5346.DBX  203.5;
      A     DB5346.DBX  201.4;
      AN    DB5346.DBX  203.1;
      AN    DB5346.DBX  203.3;
      AN    DB5346.DBX  203.4;
      =     DB5346.DBX  203.0;

// setpoint to controller ---------------
      L     DB4341.DBD 1118; // !!! insert correct SFM !!!
      T     DB5346.DBD  234;

// static value to controller ----------
      L     DB4341.DBD 1118; // !!! insert correct SFM !!!
      T     DB5346.DBD  238;

// process value to controller ----------
      L     DB5343.DBD   26; // !!! insert correct AnI !!!
      T     DB5346.DBD  254;

// low/high value to controller ---------
      L     DB5343.DBD   30; // !!! insert correct AnI !!!
      T     DB5346.DBD  218;

      L     DB5343.DBD   34; // !!! insert correct AnI !!!
      T     DB5346.DBD  222;

NETWORK
TITLE =Sequence organisation

      CLR   ;
      =     M    122.2;

// SFM supply ----------------------------------------------------------------

// analog value to SFM spare -----------------------
      L     DB5343.DBD  146;
      T     DB4341.DBD 1122; // !!! insert correct SFM !!!

// analog value to SFM spare -----------------------
      L     DB5343.DBD  266;
      T     DB4341.DBD 1122; // !!! insert correct SFM !!!

// analog value to SFM spare -----------------------
      L     DB5343.DBD  386;
      T     DB4341.DBD 1122; // !!! insert correct SFM !!!

// sequencer ----------------------------------------------------------------
      A     DB4343.DBX   43.1;
      S     DB4343.DBX   97.3;

      CALL FC    40 (
           UnitNo                   := #UnitNo);

NETWORK
TITLE =Auto / Manual

      SET   ;
      AN    M    122.2;
      JC    MODE;
      AN    M    120.1;


// assign PID mode
      S     DB5346.DBX  201.4;
      S     DB5346.DBX  201.5;


MODE: SET   ;

END_FUNCTION_BLOCK

